// Mitsubishi GX Works2 project: PLC_Group24 (1)   PLC: FX3G

// global labels: Global1
VAR_GLOBAL
  X007_Stat_Work AT X007 : BOOL;  (* יום העבודה מתחיל בלחיצה על מתג X7 *)
  Y7_Day_Work AT Y007 : BOOL;  (* נורה Y7 תשאר דלוקה לאורך כל יום העבודה *)
  X5_Emergency_switch AT X005 : BOOL;  (* לחיצה על מתג חירום X5 *)
  input_Petel AT D1110 : REAL;  (* פטל(גרם),קלט כמות פתיחה{חומר גלם} *)
  linput_Lemon AT D1120 : REAL;  (* לימון(גרם), קלט כמות פתיחה{חומר גלם} *)
  input_Stabalized AT D1130 : REAL;  (* מייצבים(גרם), קלט כמות פתיחה{חומר גלם} *)
  input_Gummy_Bears AT D1140 : INT;  (* דובי גומי(יחידות), קלט כמות פתיחה{חומר גלם} *)
  X1_Stage1_start AT X001 : BOOL;  (* בלחיצה על המתג תתבצע דגימה של Analog Input1 ויבחר סוג הגומיגם. *)
END_VAR
VAR_GLOBAL CONSTANT
  Regular_Lower_limit : INT;  (* 0 ≤ input ≤ 5          נייצר גומיגם רגיל *)
  Regular_Upper_limit : INT := 5;  (* 0 ≤ input ≤ 5          נייצר גומיגם רגיל *)
  Treat_Lower_limit : INT := 6;  (* 6 ≤ input ≤ 10       נייצר גומיגם פינוק. *)
  Treat_Upper_limit : INT := 9;  (* 6 ≤ input ≤ 10       נייצר גומיגם פינוק. *)
  TABLE1_RegularPETAL_Lemon : REAL := 35;  (* טבלה 1 -        גלידה פטל רגיל -לימון   35 גרם *)
  TABLE1_RegularPETAL_Petel : REAL := 280;  (* טבלה 1 -          גלידה פטל רגיל -פטל 280 גרם *)
  TABLE1_RegularLemon_Petel : REAL;  (* טבלה 1 -        גלידה לימון רגיל -פטל     0 גרם *)
  TABLE1_RegularLemon_Lemon : REAL := 420;  (* טבלה 1 -     גלידה לימון רגיל -לימון 420 גרם *)
  TABLE1_RegularLemon_Stabalized : REAL := 70;  (* טבלה 1 - גלידה לימון רגיל -מייצבים   70 גרם *)
  TABLE1_TreatPETAL_Petel : REAL := 385;  (* טבלה 1 -          גלידה פטל פינוק -פטל 385 גרם *)
  TABLE1_TreatPETAL_Lemon : REAL := 105;  (* טבלה 1 -       גלידה פטל פינוק -לימון  105 גרם *)
  TABLE1_TreatPETAL_Stabalized : REAL := 70;  (* טבלה 1 -  גלידה פטל פינוק -מייצבים   70  גרם *)
  TABLE1_TreatLemon_Petel : REAL;  (* טבלה 1 -       גלידה לימון פינוק -פטל   0    גרם *)
  TABLE1_TreatLemon_Lemon : REAL := 560;  (* טבלה 1 -     גלידה לימון פינוק -לימון   560 גרם *)
  TABLE1_TreatLemon_Stabalized : REAL := 140;  (* טבלה 1 - גלידה לימון פינוק -מייצבים   140 גרם *)
END_VAR
VAR_GLOBAL
  amaount_Petel AT D1115 : REAL;  (* פטל(גרם),קלט כמות פתיחה{חומר גלם} *)
  amaount_Lemon AT D1125 : REAL;  (* לימון(גרם), קלט כמות פתיחה{חומר גלם} *)
  amaount_Stabalized AT D1135 : REAL;  (* מייצבים(גרם), קלט כמות פתיחה{חומר גלם} *)
  amaount_Gummy_Bears AT D1145 : INT;  (* דובי גומי(יחידות), קלט כמות פתיחה{חומר גלם} *)
  M110_Regular_Petel AT M110 : BOOL;  (* בוליאני,בדיקת כמות פטל לייצור גלידה  רגיל *)
  M230_Treat_Stabalized AT M230 : BOOL;  (* בוליאני,בדיקת כמות מייצבים לייצור גידה פינוק *)
  M220_Treat_Lemon AT M220 : BOOL;  (* בוליאני,בדיקת כמות לימון לייצור גלידה פינוק *)
  M210_Treat_Petel AT M210 : BOOL;  (* בוליאני,בדיקת כמות פטל לייצור גלידה פינוק *)
  M120_Regularl_Lemon AT M120 : BOOL;  (* בוליאני,בדיקת כמות לימון לייצור גלידה  רגיל *)
  M250_Treat_Can_produce AT M250 : BOOL;  (* בוליאני,האם יכול לייצור גלידה פינוק *)
END_VAR
VAR_GLOBAL CONSTANT
  TABLE1_RegularPETAL_Stabalized : REAL := 35;  (* טבלה 1 -   גלידה פטל רגיל -מייצבים   35 גרם *)
END_VAR
VAR_GLOBAL
  M140_Regularl_Gummy_Bears AT M140 : BOOL;  (* בוליאני,בדיקת כמות דובי גומי לייצור גלידה  רגיל *)
  M130_Regularl_Stabalized AT M130 : BOOL;  (* בוליאני,בדיקת כמות מיצבים לייצור גלידה  רגיל *)
  M240_Treat_Gummy_Bears AT M240 : BOOL;  (* בוליאני,בדיקת כמות דובי גומי לייצור גלידה פינוק *)
END_VAR
VAR_GLOBAL CONSTANT
  TABLE2_Regular_Gummy_Bears_gr : REAL := 28;  (* טבלה 2 -        גלידה פטל רגיל -דובי גומי   28 גרם *)
  TABLE2_Treat_Gummy_Bears_gr : REAL := 70;  (* טבלה 2 -      גלידה פטל פינוק -דובי גומי   70  גרם *)
END_VAR
VAR_GLOBAL
  M100_Regular AT M100 : BOOL;  (* בוליאני,לייצר גומיגם רגיל *)
  M101_Regular_Upper AT M101 : BOOL;  (* בוליאני,לייצר גומיגם רגיל-גבול עליון *)
  M102_Regular_Lower AT M102 : BOOL;  (* בוליאני,לייצר גומיגם רגיל-גבול תחתון *)
  M202_Treat_Lower AT M202 : BOOL;  (* בוליאני,לייצר גומיגם פינוק-גבול תחתון *)
  M200_Treat AT M200 : BOOL;  (* בוליאני,לייצר גומיגם פינוק *)
  M201_Treat_Upper AT M201 : BOOL;  (* בוליאני,לייצר גומיגם פינוק-גבול עליון *)
  M150_Regular_Can_produce AT M150 : BOOL;  (* בוליאני,האם יכול לייצור גלידה  רגיל *)
END_VAR
VAR_GLOBAL CONSTANT
  Analog_Input_divader : INT := 400;  (* Analog Input התאמת ערכי החיבור בחילוק ב400 *)
END_VAR
VAR_GLOBAL
  adj_analog_input_1 AT D1105 : INT;  (* דובי גומי(יחידות), קלט כמות פתיחה{חומר גלם} *)
  Y0_Ice_Cream_In_Process AT Y000 : BOOL;  (* הכנת הגלידה נמשכת 5 שניות במהלכן נורה Y0 דולקת. *)
  M_10_Not_Enough_Resources AT M10 : BOOL;  (* חסר חומר גלם - במידה ודולק יש לעצור מיידית את הייצור *)
  TS1_Coock_Ligth AT TS1 : BOOL;  (* בוליאני,האם יכול לייצור גלידה  רגיל *)
  TC1_stap1_cook_Ice_Cream AT TC1 : BOOL;  (* טיימר של 5 שניות,שלב 1 , של הכנת הגלידה *)
END_VAR
VAR_GLOBAL CONSTANT
  Time_cook_Ice_Cream : INT := 50;  (* 5 שניות של שלב ראשון של בישול הגלידה *)
END_VAR
VAR_GLOBAL
  Container_Ice_Cream_Petel AT D1150 : REAL;  (* מיכל ההכנה,גלידת פטל(גרם) כמויות, *)
  Container_Ice_Cream_Lemon AT D1160 : REAL;  (* מיכל ההכנה,גלידת לימון(גרם) כמויות *)
  Container_Cooling_Petel AT D1170 : REAL;  (* מיכל הקירור,גלידת פטל(גרם) כמויות *)
  Container_Cooling_Lemon AT D1180 : REAL;  (* מיכל הקירור,גלידת לימון(גרם) כמויות *)
  container_Mixing AT D1190 : REAL;  (* מיכל הערבוב של הגלידות ביחד עם גלידת הפט, גלידת הלימון, והגומיגם ביחד *)
END_VAR
VAR_GLOBAL CONSTANT
  Emptying_Container : REAL;  (* ריקון המיכל לאחר שהועבר למיכל אחר *)
END_VAR
VAR_GLOBAL
  X2_Stage2_start AT X002 : BOOL;  (* ע"י לחיצה על מתג X2 הגלידה תועבר ממכלי הכנת הטעמים למכלי הקירור (מכל נפרד עבור כל טעם) ותהליך הקירור מתחיל. *)
  Y2_step2_Cooling_In_Process AT Y002 : BOOL;  (* במהלך הקירור נורה 2Y דולקת. *)
  TS2_Cooling_Ligth AT TS2 : BOOL;  (* בוליאני,האם האם מקרר את הגלידה *)
  TC2_stap2_Cooling_Ice_Cream AT TC2 : BOOL;  (* משך קירור הגלידה הוא עד 8 שניות *)
END_VAR
VAR_GLOBAL CONSTANT
  Time_Cooling_Ice_Cream : INT := 80;  (* משך קירור הגלידה הוא עד 8 שניות *)
END_VAR
VAR_GLOBAL
  X3_High_temp_switch AT X003 : BOOL;  (* או עד שחיישן הטמפרטורה X3 מצביע על טמפרטורה של 10 מעלות ומטה. *)
  Y5_step3_Mixing_In_Progress AT Y005 : BOOL;  (* משך הערבוב תלוי בסוג הגומיגם, ניתן לראות טבלה 3. בזמן הערבוב נורות Y5 ו-Y6 מהבהבות לסירוגין *)
  Y6_step3_Mixing_In_Progress AT Y006 : BOOL;  (* משך הערבוב תלוי בסוג הגומיגם, ניתן לראות טבלה 3. בזמן הערבוב נורות Y5 ו-Y6 מהבהבות לסירוגין *)
  M56_Flashing_Intermittently_Y5_6 AT M56 : BOOL;  (* בוליאני של הבהוב הורות Y5 ו- Y6 *)
  Step3_Mixing_Time AT D1300 : INT;  (* מקבל בהתאם את הערך הרצוי מטבלה 3 - בהתאם לסוג הגומיגם שייצרנו *)
  TS4_Flashing_Ligth1 AT TS4 : BOOL;  (* בוליאני,האם האם מערבב - 2 *)
  TC4_stap3_Mixing1 AT TC4 : BOOL;  (* משך קירור הגלידה הוא ערבוב תלוי בסוג הגומיגם לפי טבלה 3 *)
  TS5_Flashing_Ligth2 AT TS5 : BOOL;  (* בוליאני,האם האם מערבב - 2 *)
  TC5_stap3_Mixing2 AT TC5 : BOOL;  (* משך קירור הגלידה הוא ערבוב תלוי בסוג הגומיגם לפי טבלה 3 *)
END_VAR
VAR_GLOBAL CONSTANT
  TABLE2_Regular_Gummy_Bears_unit : INT := 28;  (* טבלה 2 -        גלידה פטל רגיל -דובי גומי   28 גרם *)
  TABLE2_Treat_Gummy_Bears_unit : INT := 70;  (* טבלה 2 -      גלידה פטל פינוק -דובי גומי   70  גרם *)
  TABLE3_Treat_Mixing_time : INT := 50;  (* טבלה 3- משך זמן הערבוב (5 שניות) כתלות בסוג הגומיגם (פינוק) *)
  TABLE3_Regular_Mixing_time : INT := 30;  (* טבלה 3- משך זמן הערבוב (3 שניות) כתלות בסוג הגומיגם (רגיל) *)
END_VAR
VAR_GLOBAL
  M300_Stage3_Sart AT M300 : BOOL;  (* התחל שלב 3 , סיום שלב 2 *)
  X4_Stage4_start AT X004 : BOOL;  (* שלב 4 	תהליך זה יתחיל ע"י הרמת מתג X4. *)
  X0_One_Cone_package AT X000 : BOOL;  (* עבור אריזת גביע גומיגם בודד יש להרים את מתג X0. *)
  Y4_step4_Pakage_7Cone_in_process AT Y004 : BOOL;  (* •	בסיום אריזת הגביע הראשון במארז, יש להדליק את נורה Y4, ובסיום אריזת המארז נורה Y4 תיכבה. *)
END_VAR
VAR_GLOBAL CONSTANT
  Step3_flashing_switch : INT := 1;  (* מקבל בהתאם את הערך הרצוי מטבלה 3 - בהתאם לסוג הגומיגם שייצרנו *)
END_VAR
VAR_GLOBAL
  TS3_Micing_time AT TS3 : BOOL;  (* בוליאני,האם האם מערבב - 2 *)
  TC3_stap3_Mixing AT TC3 : BOOL;  (* משך קירור הגלידה הוא ערבוב תלוי בסוג הגומיגם לפי טבלה 3 *)
END_VAR
VAR_GLOBAL CONSTANT
  Step4_count_7cones : INT := 7;  (* ספירה של 7 גביעים באריזת הגומיגם *)
  Step4_count_First_cones : INT := 1;  (* ספירה של ביע הראשון שנכנס לאירזה *)
END_VAR
VAR_GLOBAL
  CC1_count_First_Cones AT CC1 : BOOL;  (* ספירה של 1 גביעי גלידה *)
  CC0_count_7Cones AT CC0 : BOOL;  (* ספירה של 7 גביעי גלידה *)
  CS1_count_first_cone AT CS1 : BOOL;  (* ספירה של 1 גביעי גלידה *)
  CS0_count_7_cone AT CS0 : BOOL;  (* ספירה של 7 גביעי גלידה *)
END_VAR
VAR_GLOBAL CONSTANT
  Add_one_pack : INT := 1;  (* הוספת אריזה אחת לכמות באחסון *)
  Tourn_false : BOOL;  (* הפיכת המשתנים ל-FFALSE *)
  table2_Regular_1cone_Total_grams : REAL := 124;  (* כמות הגרם הנדרשת ליחידת גומיגם רגיל אחד (124גרם) *)
  table2_Treat_1cone_Total_grams : REAL := 190;  (* כמות הגרם הנדרשת ליחידת גומיגם רגיל אחד (190גרם) *)
  New_day_Storage_is_empty : INT;  (* יום חדש, "כל המשתנים יתאפסו וניתן יהיה להתחיל יום עבודה מחדש בלחיצה נוספת על מתג X7. " *)
END_VAR
VAR_GLOBAL
  Analog_Input_1 AT D8280 : INT;  (* Analog Input 1 – D8280 --> סוג הגומיגם יבחר כתלות בערך *)
  AnalogOutput AT D8282 : INT;  (* Analog Output – D8282 --> מספר מארזי הגומיגם שיוצרו במהלך היום ביחידות עשרוניות *)
  Total_Packs AT D1100 : INT;
END_VAR
VAR_GLOBAL CONSTANT
  adj_amaunt_Packs_To_AnalogOutpot : INT := 40;  (* הערך המותאם ליציאה האנלוגית(בהכפלה ב40) *)
END_VAR
VAR_GLOBAL
  M_20_Not_Enough_Resources AT M20 : BOOL;  (* חסר חומר גלם - שלב 4 , במידה ודולק יש לעצור מיידית את הייצור *)
END_VAR

// task Task_01 (event TRUE, interval 0, priority 31): POU_01

PROGRAM POU_01
(* structured ladder/FBD written out as ST: instructions are called as NAME(EN, inputs, outputs); _pN, _eN, _tN stand for wires *)
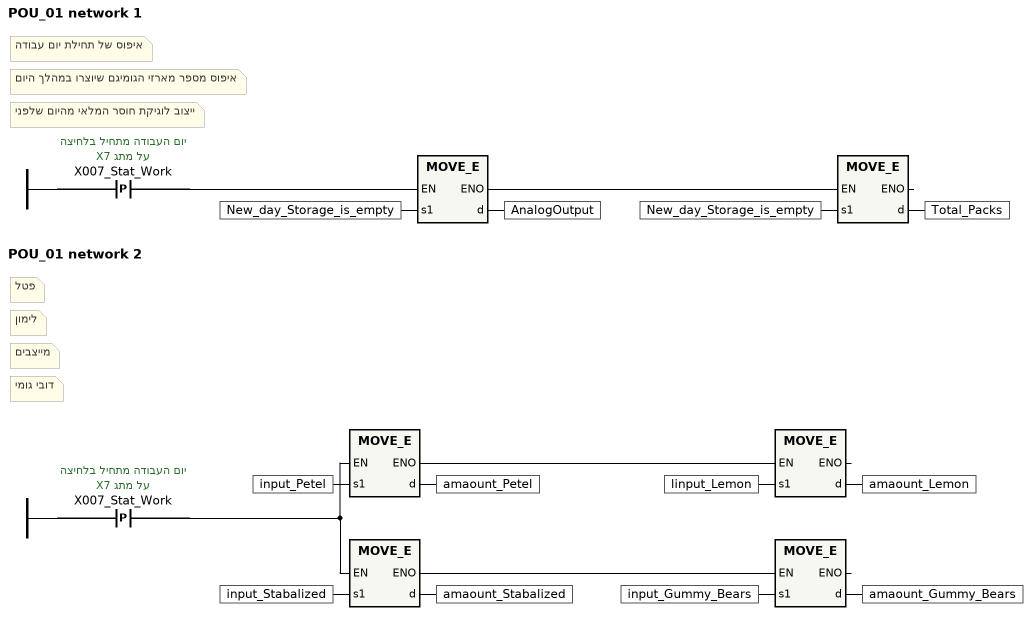
(* network 1 איפוס תחילת יום *)
(* איפוס של תחילת יום עבודה *)
(* איפוס מספר מארזי הגומיגם שיוצרו במהלך היום *)
(* ייצוב לוגיקת חוסר המלאי מהיום שלפני *)
_e1 := MOVE_E(LDP(TRUE, X007_Stat_Work), New_day_Storage_is_empty, AnalogOutput);
MOVE_E(_e1, New_day_Storage_is_empty, Total_Packs);
(* network 2 הזנת מלאי לערכים *)
(* פטל *)
(* לימון *)
(* מייצבים *)
(* דובי גומי *)
_p1 := LDP(TRUE, X007_Stat_Work);
_e2 := MOVE_E(_p1, input_Petel, amaount_Petel);
MOVE_E(_e2, linput_Lemon, amaount_Lemon);
_e3 := MOVE_E(_p1, input_Stabalized, amaount_Stabalized);
MOVE_E(_e3, input_Gummy_Bears, amaount_Gummy_Bears);
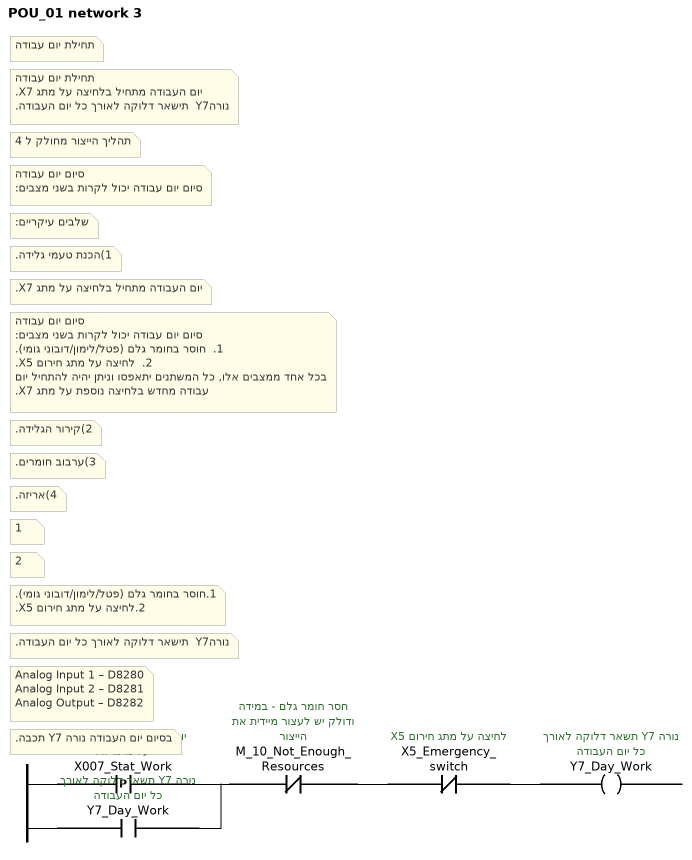
(* network 3 תחילת/סיום יום עבודה *)
(* תחילת יום עבודה *)
(* תחילת יום עבודה / יום העבודה מתחיל בלחיצה על מתג X7.   / נורהY7  תישאר דלוקה לאורך כל יום העבודה. *)
(* תהליך הייצור מחולק ל 4 *)
(* סיום יום עבודה / סיום יום עבודה יכול לקרות בשני מצבים: *)
(* שלבים עיקריים: *)
(* 1)הכנת טעמי גלידה. *)
(* יום העבודה מתחיל בלחיצה על מתג X7. *)
(* סיום יום עבודה / סיום יום עבודה יכול לקרות בשני מצבים: / 1.	חוסר בחומר גלם (פטל/לימון/דובוני גומי). / 2.	לחיצה על מתג חירום X5.  / בכל אחד ממצבים אלו, כל המשתנים יתאפסו וניתן יהיה להתחיל יום עבודה מחדש בלחיצה נוספת על מתג X7. *)
(* 2)קירור הגלידה. *)
(* 3)ערבוב חומרים. *)
(* 4)אריזה. *)
(* 1 *)
(* 2 *)
(* 1.חוסר בחומר גלם (פטל/לימון/דובוני גומי). / 2.לחיצה על מתג חירום X5. *)
(* נורהY7  תישאר דלוקה לאורך כל יום העבודה. *)
(* Analog Input 1 – D8280 / Analog Input 2 – D8281 / Analog Output – D8282 *)
(* בסיום יום העבודה נורה Y7 תכבה. *)
Y7_Day_Work := ((LDP(TRUE, X007_Stat_Work) OR Y7_Day_Work) AND NOT M_10_Not_Enough_Resources) AND NOT X5_Emergency_switch;
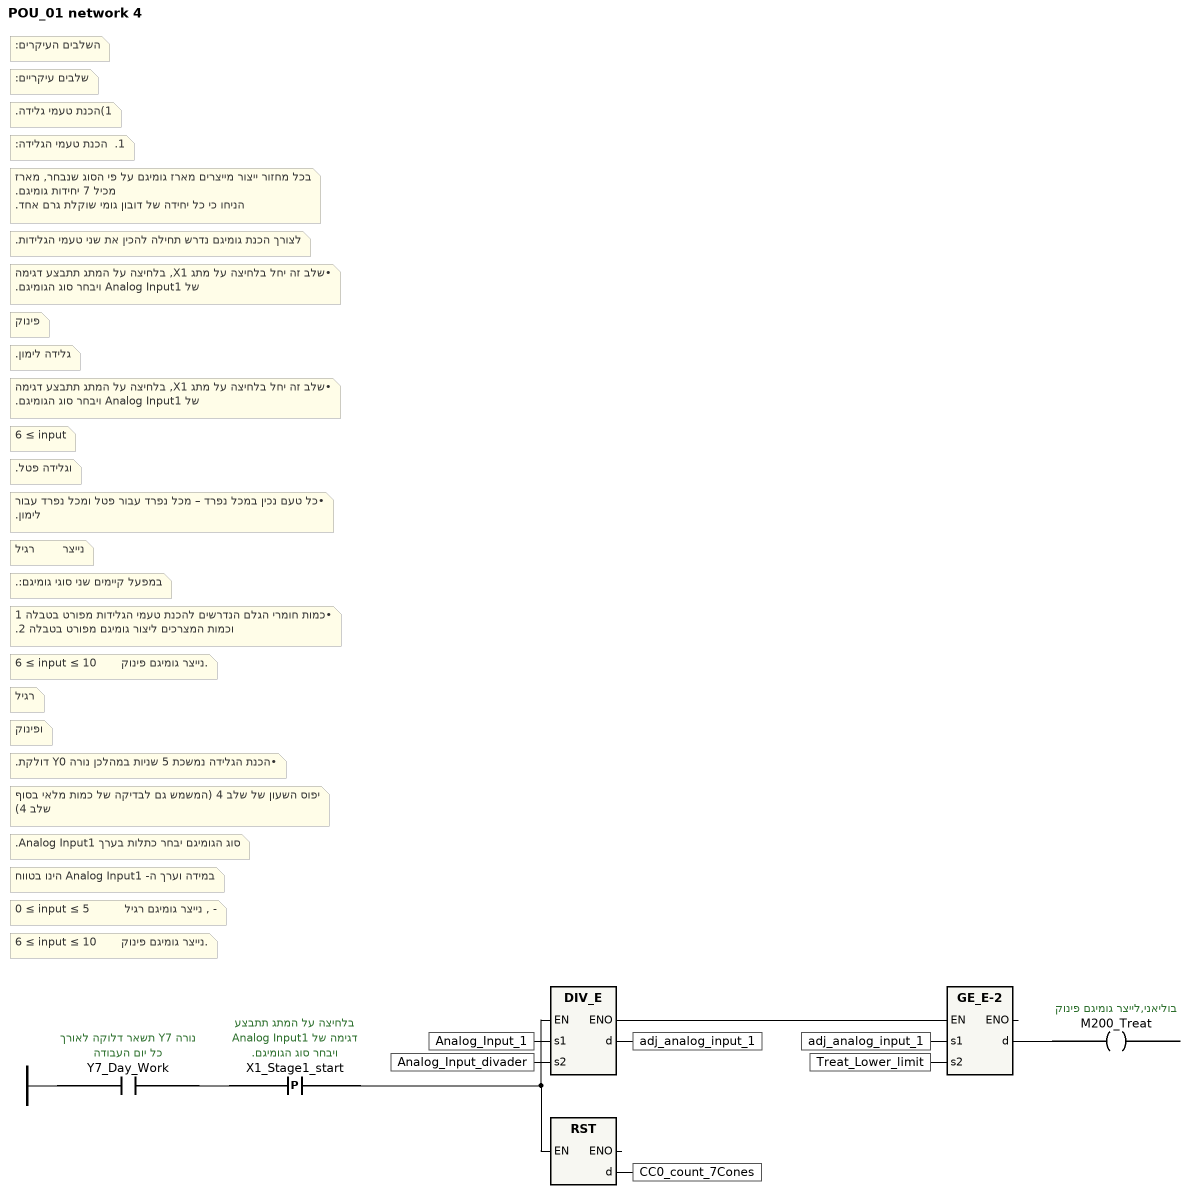
(* network 4 תחילה ובחירת סוג *)
(* השלבים העיקרים: *)
(* שלבים עיקריים: *)
(* 1)הכנת טעמי גלידה. *)
(* 1.	הכנת טעמי הגלידה: *)
(* בכל מחזור ייצור מייצרים מארז גומיגם על פי הסוג שנבחר, מארז מכיל 7 יחידות גומיגם.  / הניחו כי כל יחידה של דובון גומי שוקלת גרם אחד. *)
(* לצורך הכנת גומיגם נדרש תחילה להכין את שני טעמי הגלידות. *)
(* •שלב זה יחל בלחיצה על מתג X1, בלחיצה על המתג תתבצע דגימה של Analog Input1 ויבחר סוג הגומיגם. *)
(* פינוק *)
(* גלידה לימון. *)
(* •שלב זה יחל בלחיצה על מתג X1, בלחיצה על המתג תתבצע דגימה של Analog Input1 ויבחר סוג הגומיגם. *)
(* 6 ≤ input *)
(* וגלידה פטל. *)
(* •כל טעם נכין במכל נפרד – מכל נפרד עבור פטל ומכל נפרד עבור לימון. *)
(* נייצר        רגיל *)
(* במפעל קיימים שני סוגי גומיגם:. *)
(* •כמות חומרי הגלם הנדרשים להכנת טעמי הגלידות מפורט בטבלה 1 וכמות המצרכים ליצור גומיגם מפורט בטבלה 2. *)
(* 6 ≤ input ≤ 10       נייצר גומיגם פינוק. *)
(* רגיל *)
(* ופינוק *)
(* •הכנת הגלידה נמשכת 5 שניות במהלכן נורה Y0 דולקת. *)
(* יפוס השעון של שלב 4 (המשמש גם לבדיקה של כמות מלאי בסוף שלב 4) *)
(* סוג הגומיגם יבחר כתלות בערך Analog Input1. *)
(* במידה וערך ה- Analog Input1 הינו בטווח *)
(* 0 ≤ input ≤ 5          נייצר גומיגם רגיל , - *)
(* 6 ≤ input ≤ 10       נייצר גומיגם פינוק. *)
_p1 := Y7_Day_Work AND LDP(TRUE, X1_Stage1_start);
_e2 := DIV_E(_p1, Analog_Input_1, Analog_Input_divader, adj_analog_input_1);
GE_E(_e2, adj_analog_input_1, Treat_Lower_limit, _t3);
M200_Treat := _t3;
RST(_p1, CC0_count_7Cones);
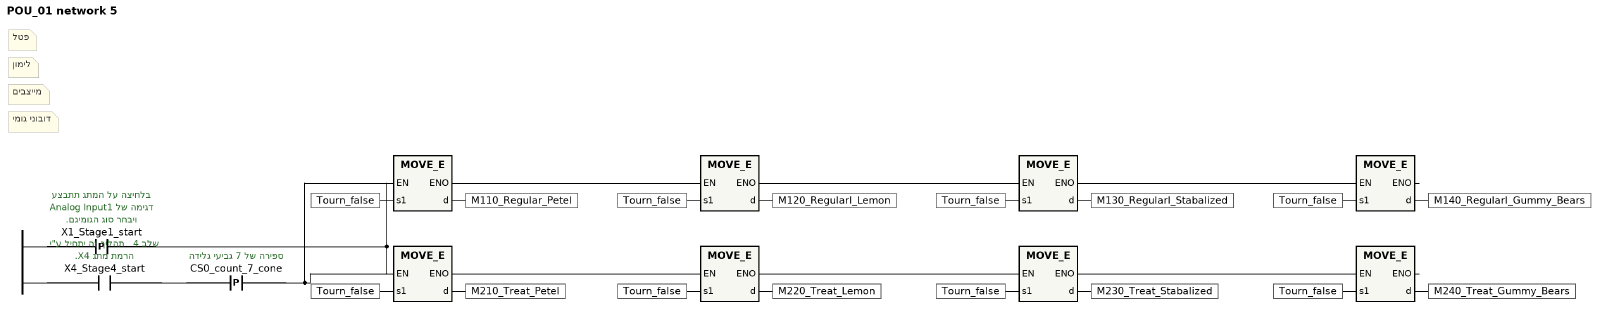
(* network 5 *)
(* פטל *)
(* לימון *)
(* מייצבים *)
(* דובוני גומי *)
_p1 := LDP(TRUE, X1_Stage1_start) OR (X4_Stage4_start AND LDP(TRUE, CS0_count_7_cone));
_e2 := MOVE_E(_p1, Tourn_false, M110_Regular_Petel);
_e3 := MOVE_E(_e2, Tourn_false, M120_Regularl_Lemon);
_e4 := MOVE_E(_e3, Tourn_false, M130_Regularl_Stabalized);
MOVE_E(_e4, Tourn_false, M140_Regularl_Gummy_Bears);
_e5 := MOVE_E(_p1, Tourn_false, M210_Treat_Petel);
_e6 := MOVE_E(_e5, Tourn_false, M220_Treat_Lemon);
_e7 := MOVE_E(_e6, Tourn_false, M230_Treat_Stabalized);
MOVE_E(_e7, Tourn_false, M240_Treat_Gummy_Bears);
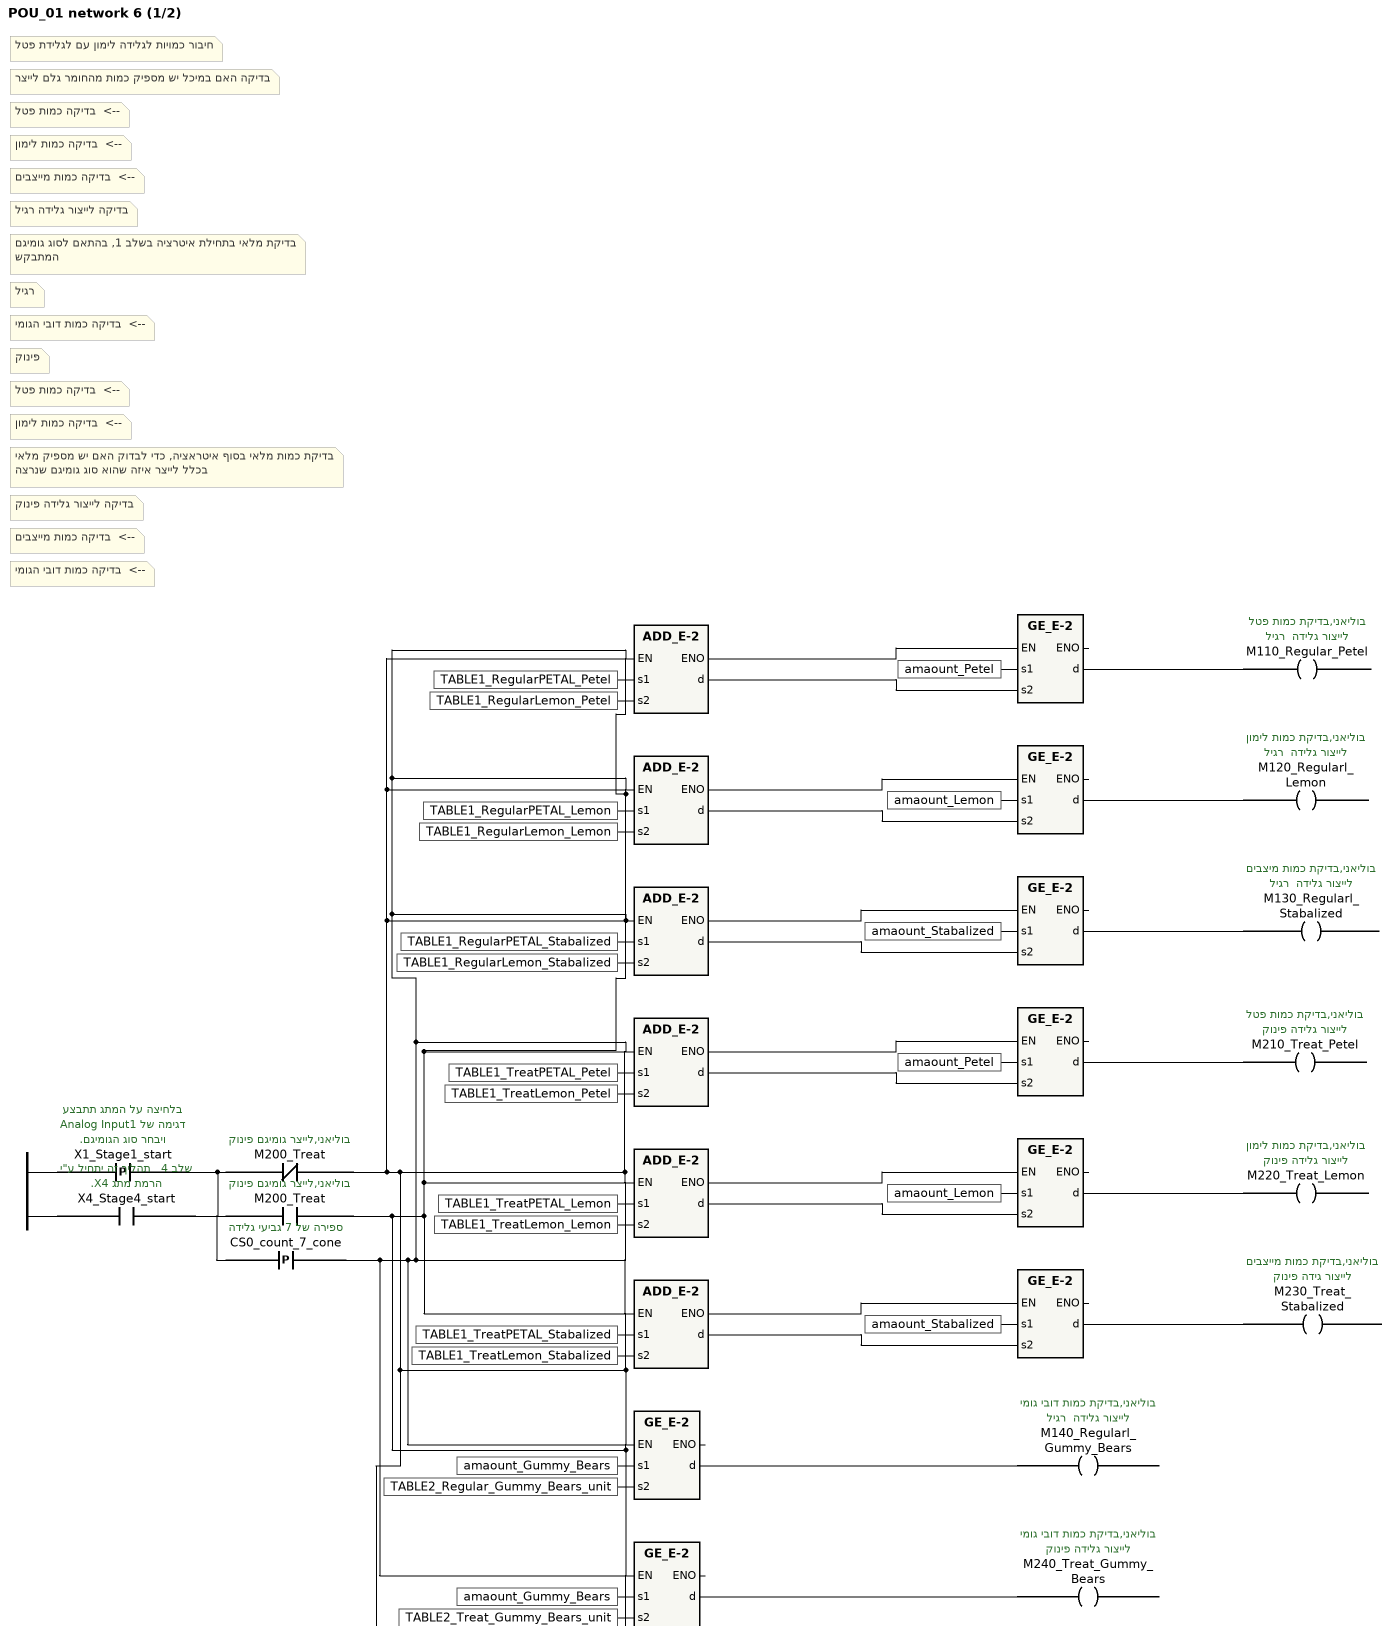
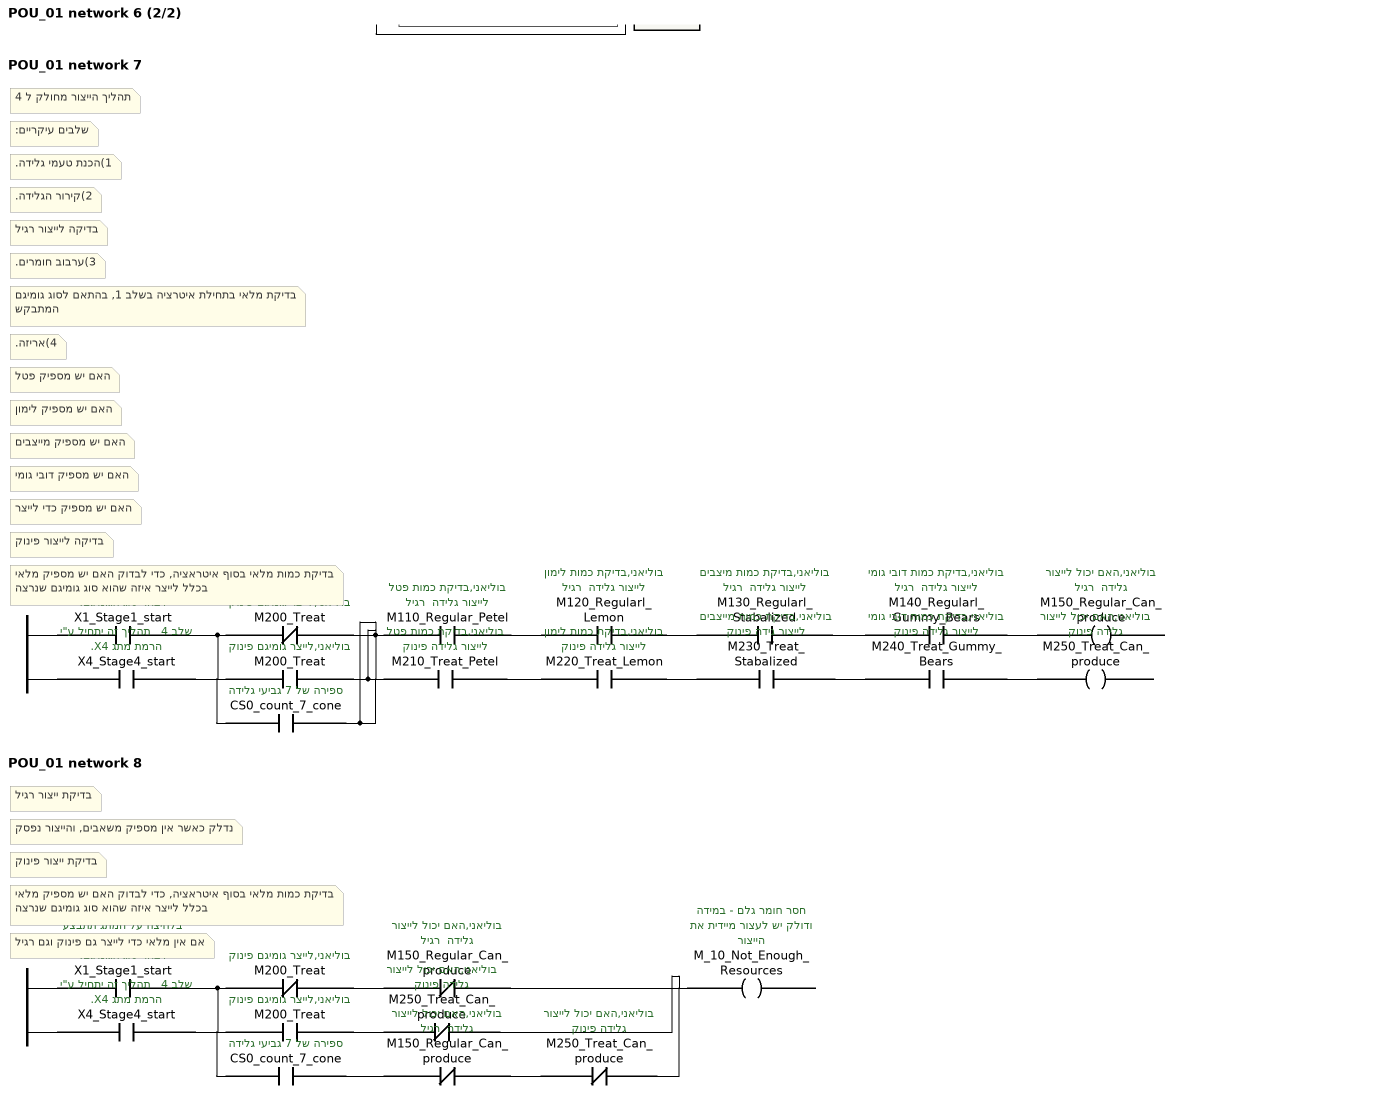
(* network 6 *)
(* חיבור כמויות לגלידה לימון עם לגלידת פטל *)
(* בדיקה האם במיכל יש מספיק כמות מהחומר גלם לייצר *)
(* -->  בדיקה כמות פטל *)
(* -->  בדיקה כמות לימון *)
(* -->  בדיקה כמות מייצבים *)
(* בדיקה לייצור גלידה רגיל *)
(* בדיקת מלאי בתחילת איטרציה בשלב 1, בהתאם לסוג גומיגם המתבקש *)
(* רגיל *)
(* -->  בדיקה כמות דובי הגומי *)
(* פינוק *)
(* -->  בדיקה כמות פטל *)
(* -->  בדיקה כמות לימון *)
(* בדיקת כמות מלאי בסוף איטראציה, כדי לבדוק האם יש מספיק מלאי בכלל לייצר איזה שהוא סוג גומיגם שנרצה *)
(* בדיקה לייצור גלידה פינוק *)
(* -->  בדיקה כמות מייצבים *)
(* -->  בדיקה כמות דובי הגומי *)
_p1 := LDP(TRUE, X1_Stage1_start);
_p2 := (_p1 AND NOT M200_Treat) OR (_p1 AND M200_Treat) OR (X4_Stage4_start AND LDP(TRUE, CS0_count_7_cone));
_e4 := ADD_E(_p2, TABLE1_RegularPETAL_Petel, TABLE1_RegularLemon_Petel, _t3);
GE_E(_e4, amaount_Petel, _t3, _t5);
M110_Regular_Petel := _t5;
_e7 := ADD_E(_p2, TABLE1_RegularPETAL_Lemon, TABLE1_RegularLemon_Lemon, _t6);
GE_E(_e7, amaount_Lemon, _t6, _t8);
M120_Regularl_Lemon := _t8;
_e10 := ADD_E(_p2, TABLE1_RegularPETAL_Stabalized, TABLE1_RegularLemon_Stabalized, _t9);
GE_E(_e10, amaount_Stabalized, _t9, _t11);
M130_Regularl_Stabalized := _t11;
GE_E(_p2, amaount_Gummy_Bears, TABLE2_Regular_Gummy_Bears_unit, _t12);
M140_Regularl_Gummy_Bears := _t12;
_e14 := ADD_E(_p2, TABLE1_TreatPETAL_Petel, TABLE1_TreatLemon_Petel, _t13);
GE_E(_e14, amaount_Petel, _t13, _t15);
M210_Treat_Petel := _t15;
_e17 := ADD_E(_p2, TABLE1_TreatPETAL_Lemon, TABLE1_TreatLemon_Lemon, _t16);
GE_E(_e17, amaount_Lemon, _t16, _t18);
M220_Treat_Lemon := _t18;
_e20 := ADD_E(_p2, TABLE1_TreatPETAL_Stabalized, TABLE1_TreatLemon_Stabalized, _t19);
GE_E(_e20, amaount_Stabalized, _t19, _t21);
M230_Treat_Stabalized := _t21;
GE_E(_p2, amaount_Gummy_Bears, TABLE2_Treat_Gummy_Bears_unit, _t22);
M240_Treat_Gummy_Bears := _t22;
(* network 7 *)
(* תהליך הייצור מחולק ל 4 *)
(* שלבים עיקריים: *)
(* 1)הכנת טעמי גלידה. *)
(* 2)קירור הגלידה. *)
(* בדיקה לייצור רגיל *)
(* 3)ערבוב חומרים. *)
(* בדיקת מלאי בתחילת איטרציה בשלב 1, בהתאם לסוג גומיגם המתבקש *)
(* 4)אריזה. *)
(* האם יש מספיק פטל *)
(* האם יש מספיק לימון *)
(* האם יש מספיק מייצבים *)
(* האם יש מספיק דובי גומי *)
(* האם יש מספיק כדי לייצר *)
(* בדיקה לייצור פינוק *)
(* בדיקת כמות מלאי בסוף איטראציה, כדי לבדוק האם יש מספיק מלאי בכלל לייצר איזה שהוא סוג גומיגם שנרצה *)
_p1 := (X1_Stage1_start AND NOT M200_Treat) OR (X1_Stage1_start AND M200_Treat) OR (X4_Stage4_start AND CS0_count_7_cone);
M150_Regular_Can_produce := _p1 AND M110_Regular_Petel AND M120_Regularl_Lemon AND M130_Regularl_Stabalized AND M140_Regularl_Gummy_Bears;
M250_Treat_Can_produce := _p1 AND M210_Treat_Petel AND M220_Treat_Lemon AND M230_Treat_Stabalized AND M240_Treat_Gummy_Bears;
(* network 8 *)
(* בדיקת ייצור רגיל *)
(* נדלק כאשר אין מספיק משאבים, והייצור נפסק *)
(* בדיקת ייצור פינוק *)
(* בדיקת כמות מלאי בסוף איטראציה, כדי לבדוק האם יש מספיק מלאי בכלל לייצר איזה שהוא סוג גומיגם שנרצה *)
(* אם אין מלאי כדי לייצר גם פינוק וגם רגיל *)
M_10_Not_Enough_Resources := (X1_Stage1_start AND NOT M200_Treat AND NOT M150_Regular_Can_produce) OR (X1_Stage1_start AND M200_Treat AND NOT M250_Treat_Can_produce) OR (X4_Stage4_start AND CS0_count_7_cone AND NOT M150_Regular_Can_produce AND NOT M250_Treat_Can_produce);
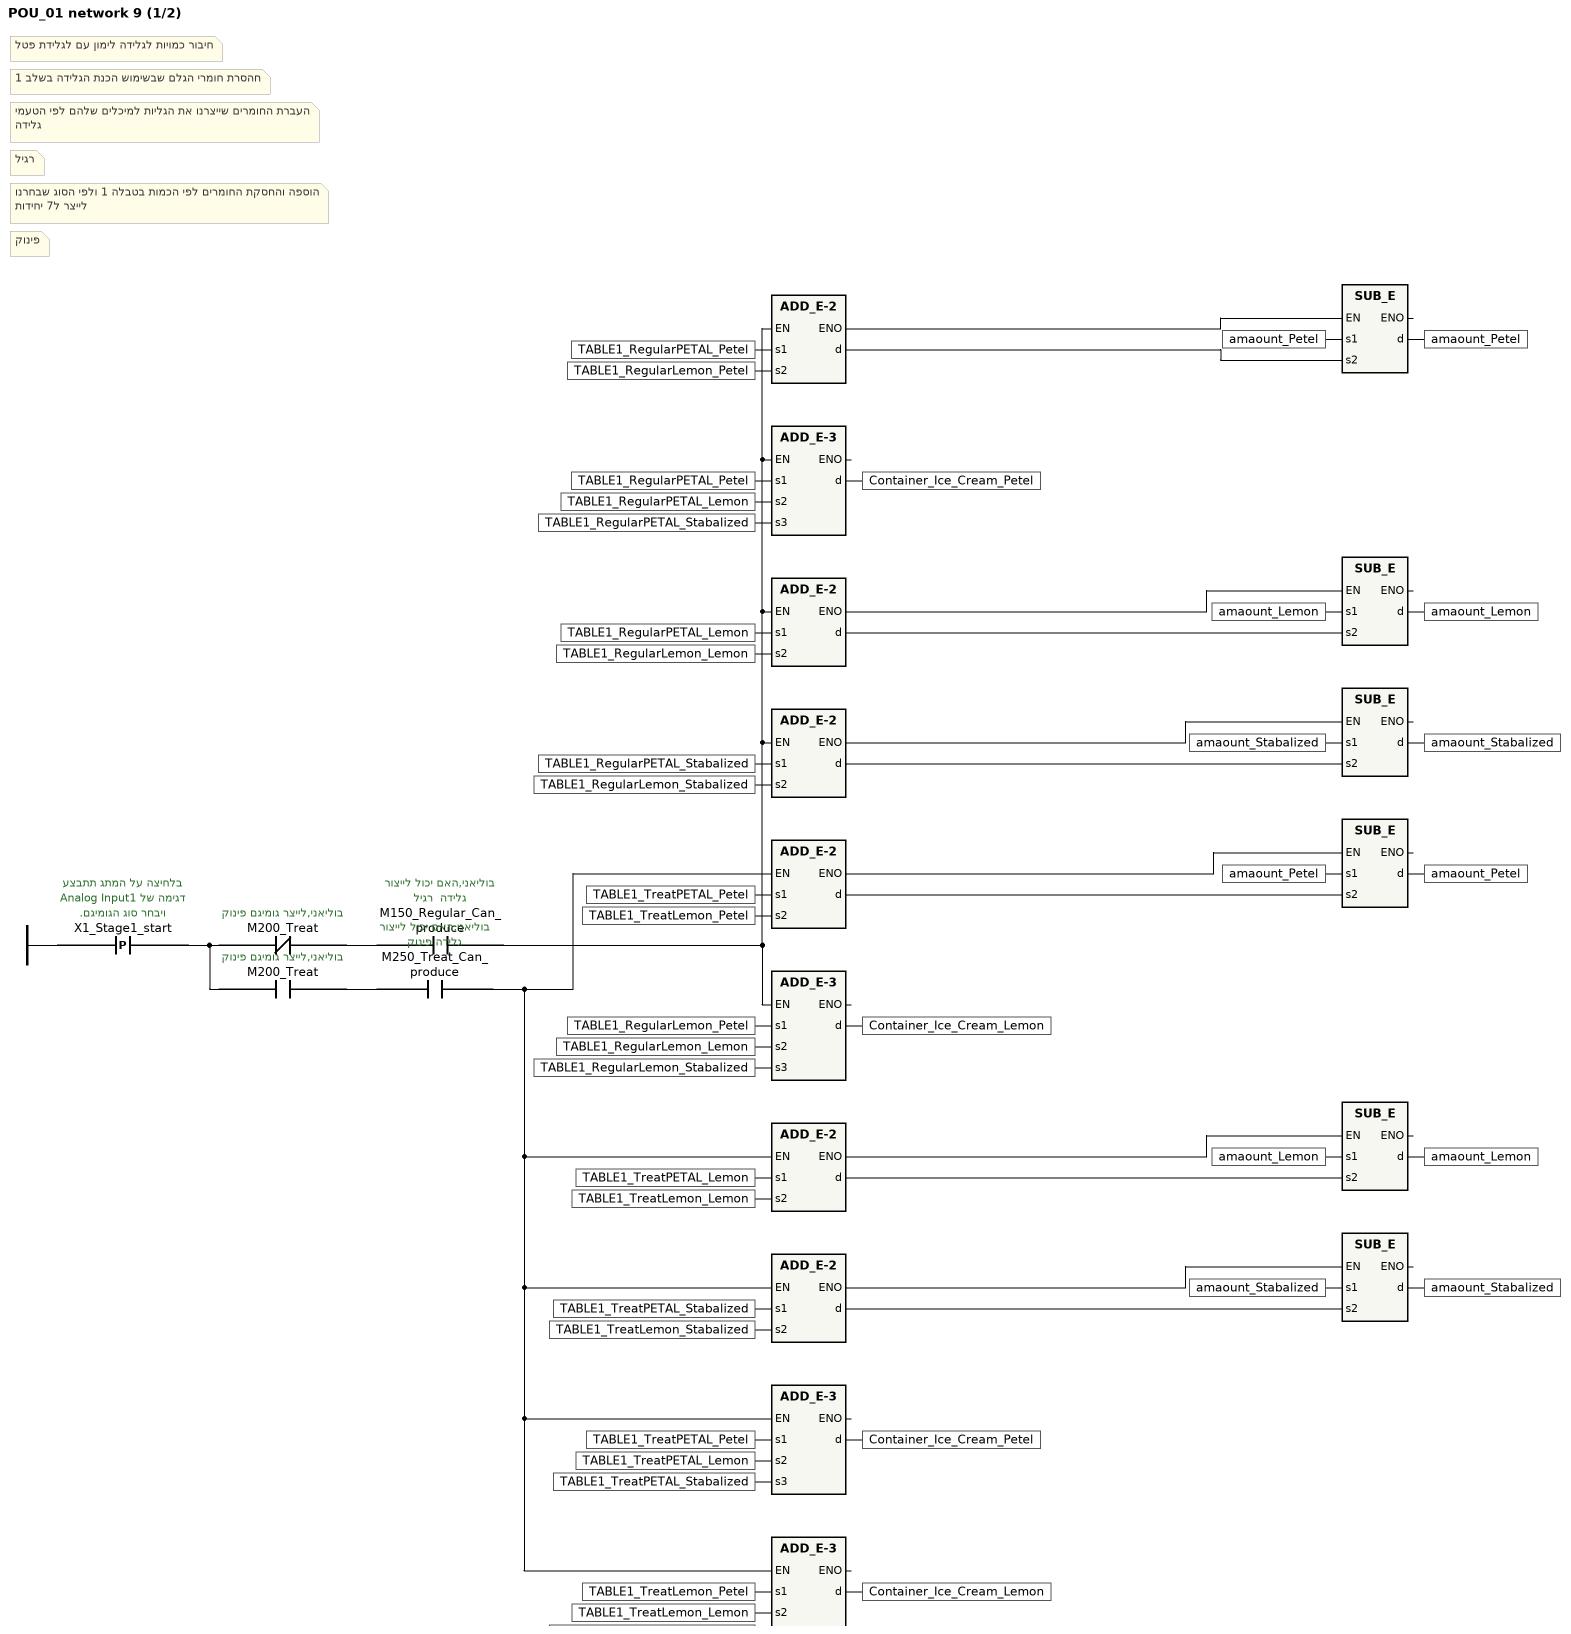
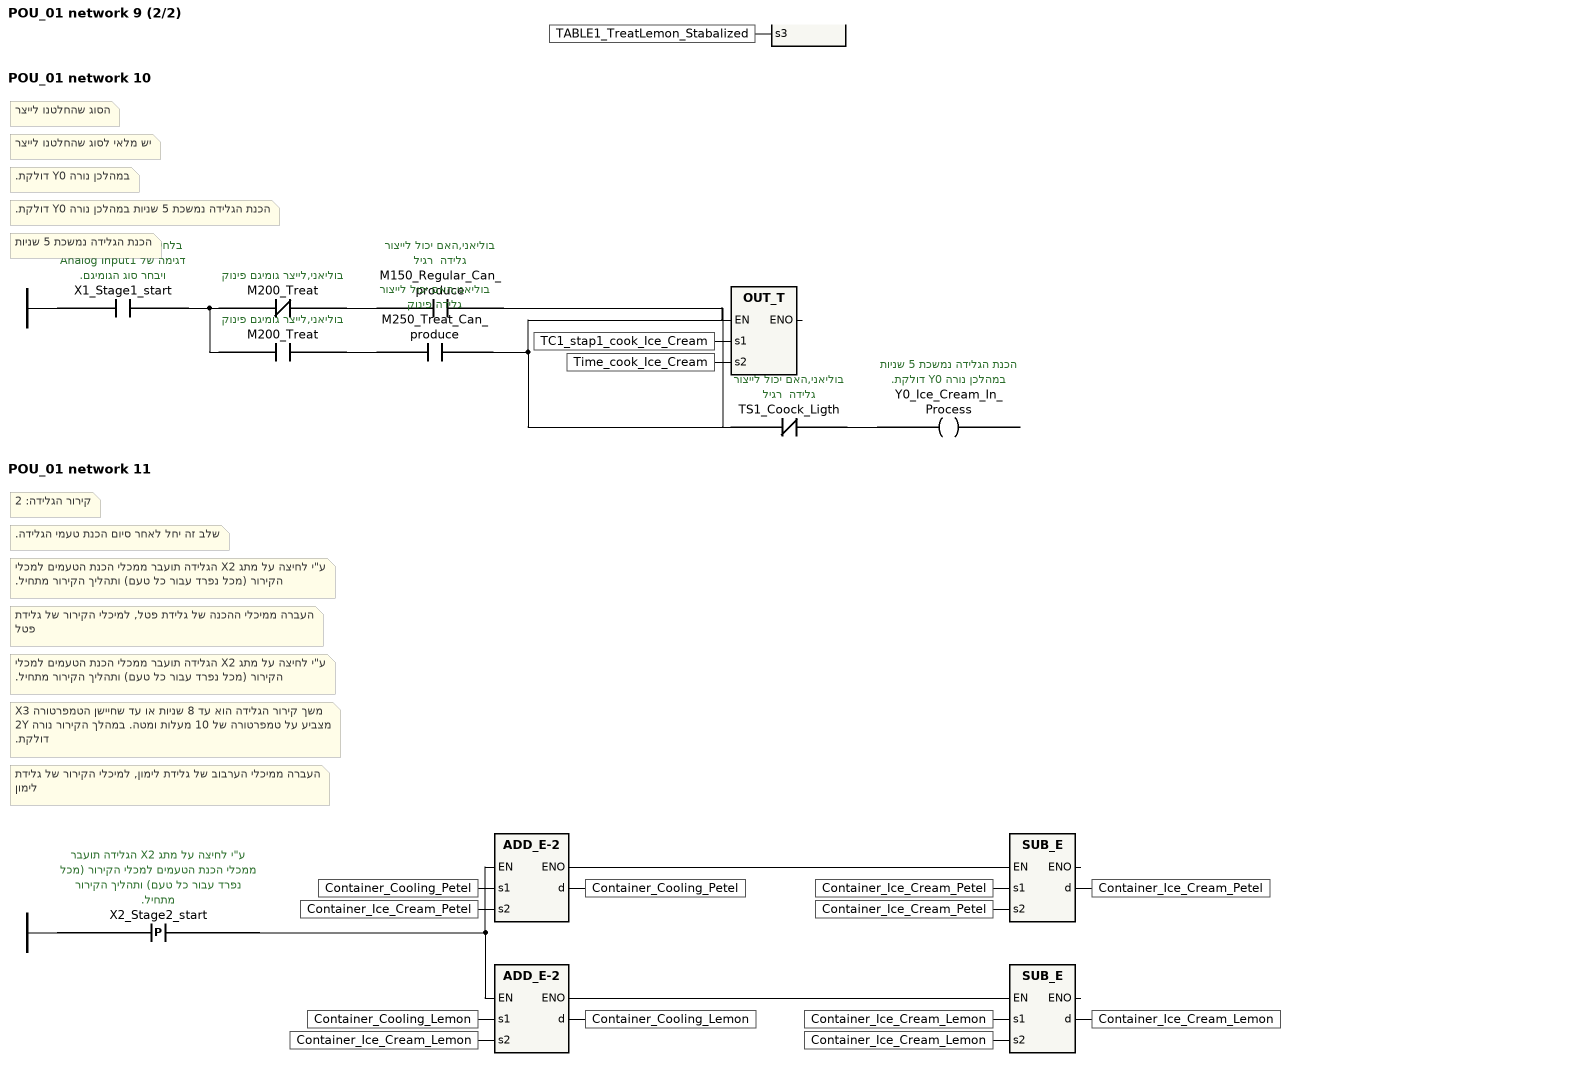
(* network 9 *)
(* חיבור כמויות לגלידה לימון עם לגלידת פטל *)
(* חהסרת חומרי הגלם שבשימוש הכנת הגלידה בשלב 1 *)
(* העברת החומרים שייצרנו את הגליות למיכלים שלהם לפי הטעמי גלידה *)
(* רגיל *)
(* הוספה והחסקת החומרים לפי הכמות בטבלה 1 ולפי הסוג שבחרנו לייצר ל7 יחידות *)
(* פינוק *)
_p1 := LDP(TRUE, X1_Stage1_start);
_p2 := _p1 AND NOT M200_Treat AND M150_Regular_Can_produce;
_e4 := ADD_E(_p2, TABLE1_RegularPETAL_Petel, TABLE1_RegularLemon_Petel, _t3);
SUB_E(_e4, amaount_Petel, _t3, amaount_Petel);
ADD_E(_p2, TABLE1_RegularPETAL_Petel, TABLE1_RegularPETAL_Lemon, TABLE1_RegularPETAL_Stabalized, Container_Ice_Cream_Petel);
_e6 := ADD_E(_p2, TABLE1_RegularPETAL_Lemon, TABLE1_RegularLemon_Lemon, _t5);
SUB_E(_e6, amaount_Lemon, _t5, amaount_Lemon);
ADD_E(_p2, TABLE1_RegularLemon_Petel, TABLE1_RegularLemon_Lemon, TABLE1_RegularLemon_Stabalized, Container_Ice_Cream_Lemon);
_e8 := ADD_E(_p2, TABLE1_RegularPETAL_Stabalized, TABLE1_RegularLemon_Stabalized, _t7);
SUB_E(_e8, amaount_Stabalized, _t7, amaount_Stabalized);
_p9 := _p1 AND M200_Treat AND M250_Treat_Can_produce;
_e11 := ADD_E(_p9, TABLE1_TreatPETAL_Petel, TABLE1_TreatLemon_Petel, _t10);
SUB_E(_e11, amaount_Petel, _t10, amaount_Petel);
ADD_E(_p9, TABLE1_TreatPETAL_Petel, TABLE1_TreatPETAL_Lemon, TABLE1_TreatPETAL_Stabalized, Container_Ice_Cream_Petel);
_e13 := ADD_E(_p9, TABLE1_TreatPETAL_Lemon, TABLE1_TreatLemon_Lemon, _t12);
SUB_E(_e13, amaount_Lemon, _t12, amaount_Lemon);
ADD_E(_p9, TABLE1_TreatLemon_Petel, TABLE1_TreatLemon_Lemon, TABLE1_TreatLemon_Stabalized, Container_Ice_Cream_Lemon);
_e15 := ADD_E(_p9, TABLE1_TreatPETAL_Stabalized, TABLE1_TreatLemon_Stabalized, _t14);
SUB_E(_e15, amaount_Stabalized, _t14, amaount_Stabalized);
(* network 10 *)
(* הסוג שהחלטנו לייצר *)
(* יש מלאי לסוג שהחלטנו לייצר *)
(* במהלכן נורה Y0 דולקת. *)
(* הכנת הגלידה נמשכת 5 שניות במהלכן נורה Y0 דולקת. *)
(* הכנת הגלידה נמשכת 5 שניות *)
_p1 := (X1_Stage1_start AND NOT M200_Treat AND M150_Regular_Can_produce) OR (X1_Stage1_start AND M200_Treat AND M250_Treat_Can_produce);
Y0_Ice_Cream_In_Process := _p1 AND NOT TS1_Coock_Ligth;
OUT_T(_p1, TC1_stap1_cook_Ice_Cream, Time_cook_Ice_Cream);
(* network 11 שלב 2 *)
(* קירור הגלידה: 2 *)
(* שלב זה יחל לאחר סיום הכנת טעמי הגלידה. *)
(* ע"י לחיצה על מתג X2 הגלידה תועבר ממכלי הכנת הטעמים למכלי הקירור (מכל נפרד עבור כל טעם) ותהליך הקירור מתחיל. *)
(* העברה ממיכלי ההכנה של גלידת פטל, למיכלי הקירור של גלידת פטל *)
(* ע"י לחיצה על מתג X2 הגלידה תועבר ממכלי הכנת הטעמים למכלי הקירור (מכל נפרד עבור כל טעם) ותהליך הקירור מתחיל. *)
(* משך קירור הגלידה הוא עד 8 שניות או עד שחיישן הטמפרטורה X3 מצביע על טמפרטורה של 10 מעלות ומטה. במהלך הקירור נורה 2Y דולקת. *)
(* העברה ממיכלי הערבוב של גלידת לימון, למיכלי הקירור של גלידת לימון *)
_p1 := LDP(TRUE, X2_Stage2_start);
_e2 := ADD_E(_p1, Container_Cooling_Petel, Container_Ice_Cream_Petel, Container_Cooling_Petel);
SUB_E(_e2, Container_Ice_Cream_Petel, Container_Ice_Cream_Petel, Container_Ice_Cream_Petel);
_e3 := ADD_E(_p1, Container_Cooling_Lemon, Container_Ice_Cream_Lemon, Container_Cooling_Lemon);
SUB_E(_e3, Container_Ice_Cream_Lemon, Container_Ice_Cream_Lemon, Container_Ice_Cream_Lemon);
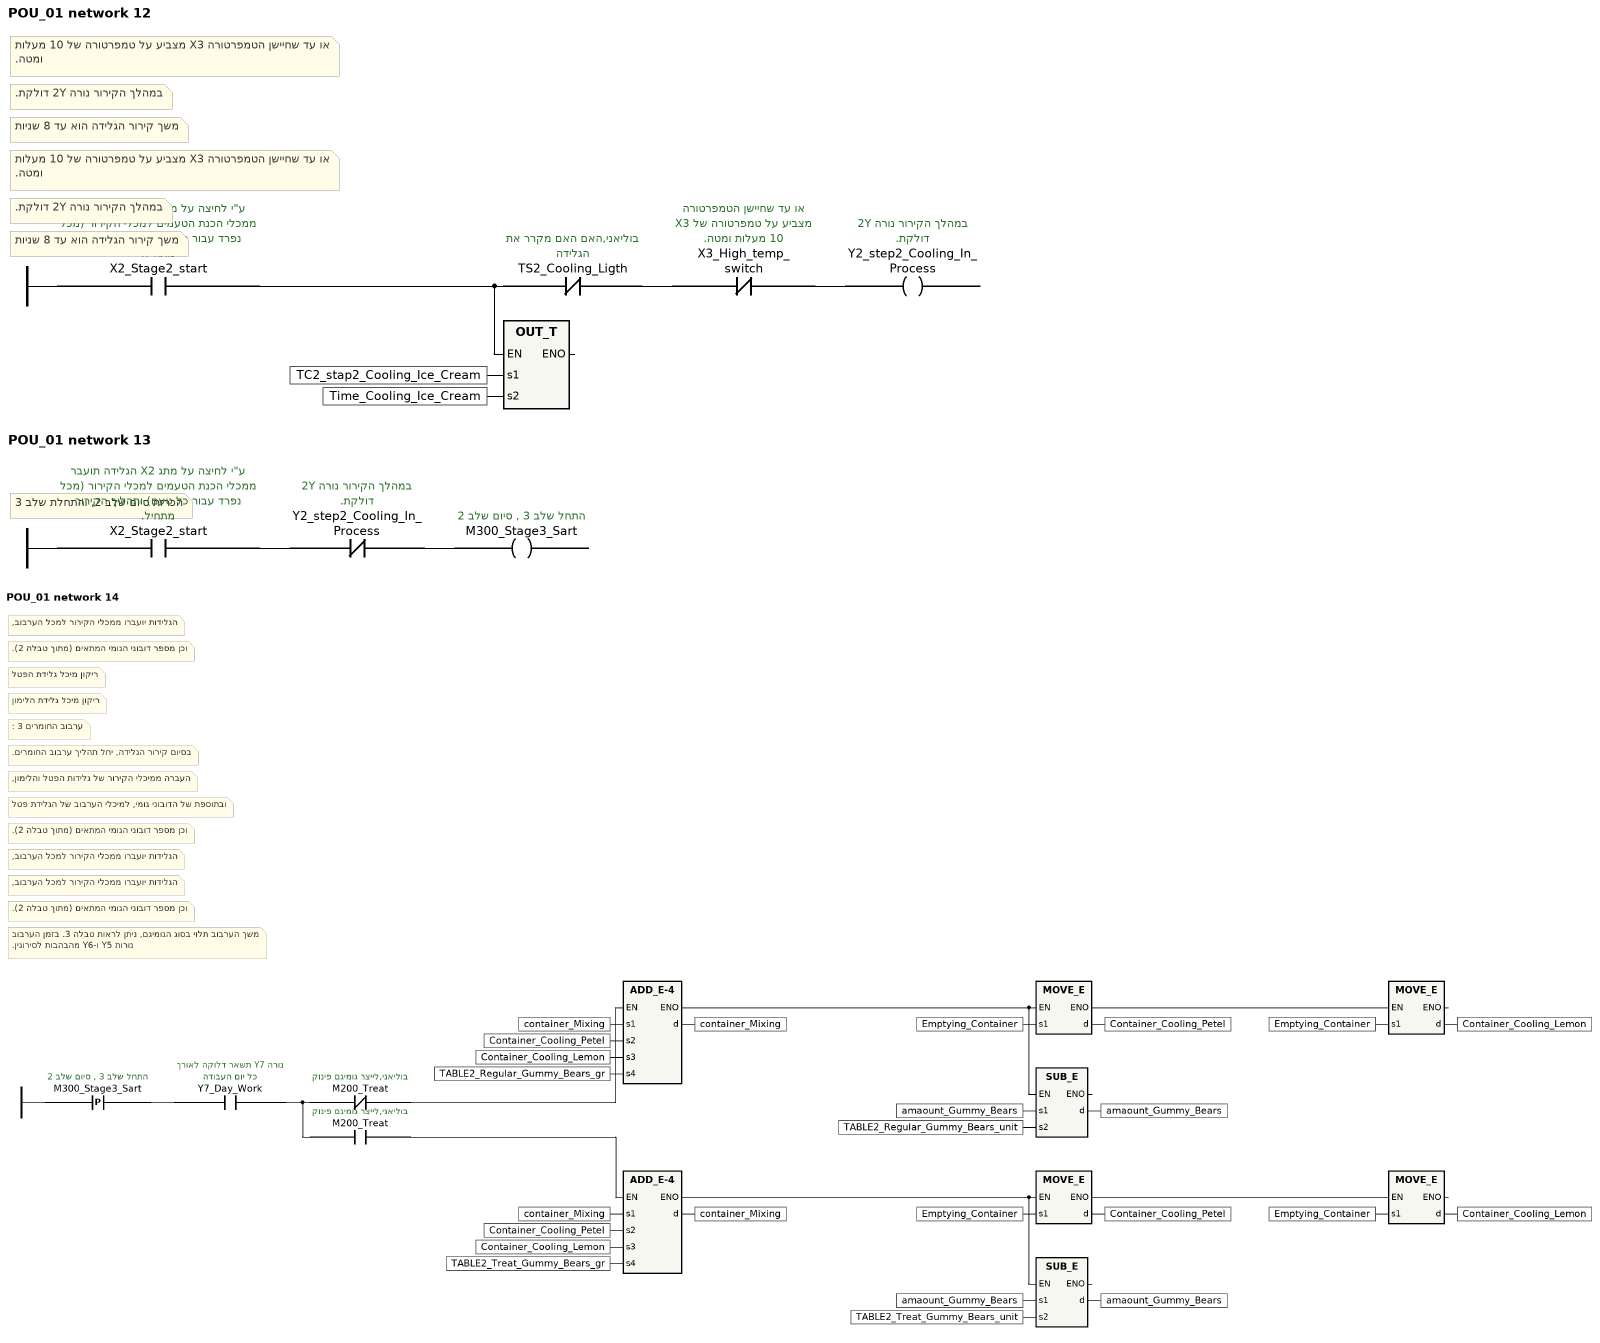
(* network 12 *)
(* או עד שחיישן הטמפרטורה X3 מצביע על טמפרטורה של 10 מעלות ומטה. *)
(* במהלך הקירור נורה 2Y דולקת. *)
(* משך קירור הגלידה הוא עד 8 שניות *)
(* או עד שחיישן הטמפרטורה X3 מצביע על טמפרטורה של 10 מעלות ומטה. *)
(* במהלך הקירור נורה 2Y דולקת. *)
(* משך קירור הגלידה הוא עד 8 שניות *)
Y2_step2_Cooling_In_Process := X2_Stage2_start AND NOT TS2_Cooling_Ligth AND NOT X3_High_temp_switch;
OUT_T(X2_Stage2_start, TC2_stap2_Cooling_Ice_Cream, Time_Cooling_Ice_Cream);
(* network 13 *)
(* הכרזת סיום שלב 2, והתחלת שלב 3 *)
M300_Stage3_Sart := X2_Stage2_start AND NOT Y2_step2_Cooling_In_Process;
(* network 14 שלב 3 *)
(* הגלידות יועברו ממכלי הקירור למכל הערבוב, *)
(* וכן מספר דובוני הגומי המתאים (מתוך טבלה 2). *)
(* ריקון מיכל גלידת הפטל *)
(* ריקון מיכל גלידת הלימון *)
(* ערבוב החומרים 3 : *)
(* בסיום קירור הגלידה, יחל תהליך ערבוב החומרים. *)
(* העברה ממיכלי הקירור של גלידות הפטל והלימון, *)
(* ובתוספת של הדובוני גומי, למיכלי הערבוב של הגלידת פטל *)
(* וכן מספר דובוני הגומי המתאים (מתוך טבלה 2). *)
(* הגלידות יועברו ממכלי הקירור למכל הערבוב, *)
(* הגלידות יועברו ממכלי הקירור למכל הערבוב, *)
(* וכן מספר דובוני הגומי המתאים (מתוך טבלה 2). *)
(* משך הערבוב תלוי בסוג הגומיגם, ניתן לראות טבלה 3. בזמן הערבוב נורות Y5 ו-Y6 מהבהבות לסירוגין. *)
_p1 := LDP(TRUE, M300_Stage3_Sart) AND Y7_Day_Work;
_e2 := ADD_E(_p1 AND NOT M200_Treat, container_Mixing, Container_Cooling_Petel, Container_Cooling_Lemon, TABLE2_Regular_Gummy_Bears_gr, container_Mixing);
_e3 := MOVE_E(_e2, Emptying_Container, Container_Cooling_Petel);
MOVE_E(_e3, Emptying_Container, Container_Cooling_Lemon);
SUB_E(_e2, amaount_Gummy_Bears, TABLE2_Regular_Gummy_Bears_unit, amaount_Gummy_Bears);
_e4 := ADD_E(_p1 AND M200_Treat, container_Mixing, Container_Cooling_Petel, Container_Cooling_Lemon, TABLE2_Treat_Gummy_Bears_gr, container_Mixing);
_e5 := MOVE_E(_e4, Emptying_Container, Container_Cooling_Petel);
MOVE_E(_e5, Emptying_Container, Container_Cooling_Lemon);
SUB_E(_e4, amaount_Gummy_Bears, TABLE2_Treat_Gummy_Bears_unit, amaount_Gummy_Bears);
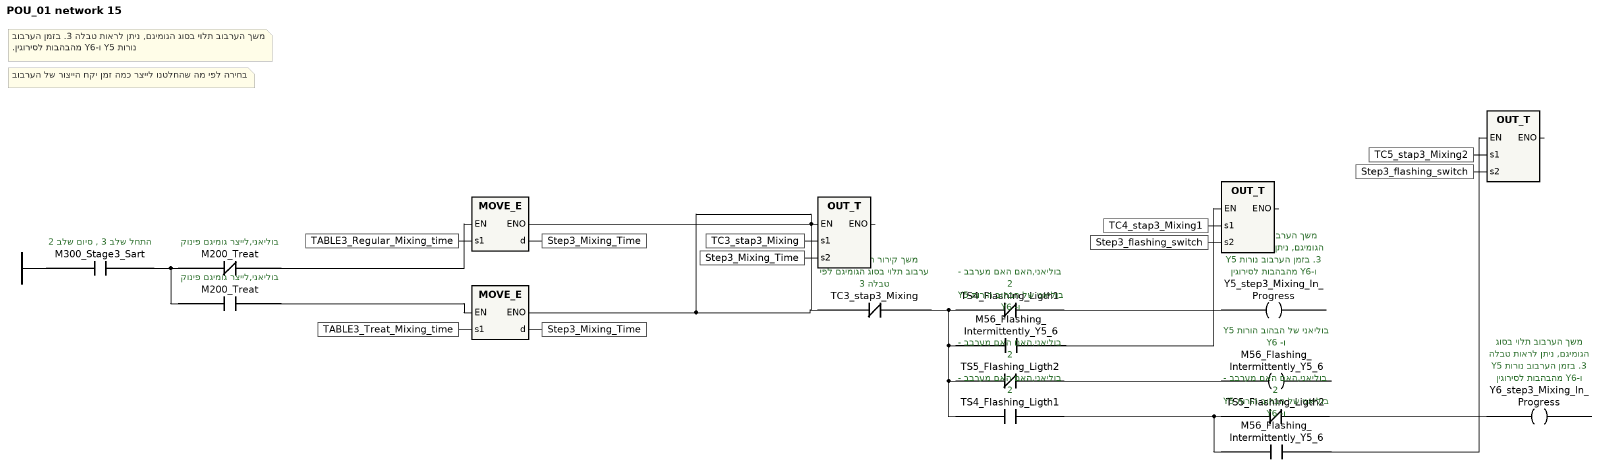
(* network 15 *)
(* משך הערבוב תלוי בסוג הגומיגם, ניתן לראות טבלה 3. בזמן הערבוב נורות Y5 ו-Y6 מהבהבות לסירוגין. *)
(* בחירה לפי מה שהחלטנו לייצר כמה זמן יקח הייצור של הערבוב *)
_e1 := MOVE_E(M300_Stage3_Sart AND NOT M200_Treat, TABLE3_Regular_Mixing_time, Step3_Mixing_Time);
_e2 := MOVE_E(M300_Stage3_Sart AND M200_Treat, TABLE3_Treat_Mixing_time, Step3_Mixing_Time);
_p3 := _e1 OR _e2;
_p4 := _p3 AND NOT TC3_stap3_Mixing;
Y5_step3_Mixing_In_Progress := _p4 AND NOT TS4_Flashing_Ligth1;
OUT_T(_p4 AND M56_Flashing_Intermittently_Y5_6, TC4_stap3_Mixing1, Step3_flashing_switch);
M56_Flashing_Intermittently_Y5_6 := _p4 AND NOT TS5_Flashing_Ligth2;
OUT_T(_p3, TC3_stap3_Mixing, Step3_Mixing_Time);
_p5 := _p4 AND TS4_Flashing_Ligth1;
Y6_step3_Mixing_In_Progress := _p5 AND NOT TS5_Flashing_Ligth2;
OUT_T(_p5 AND M56_Flashing_Intermittently_Y5_6, TC5_stap3_Mixing2, Step3_flashing_switch);
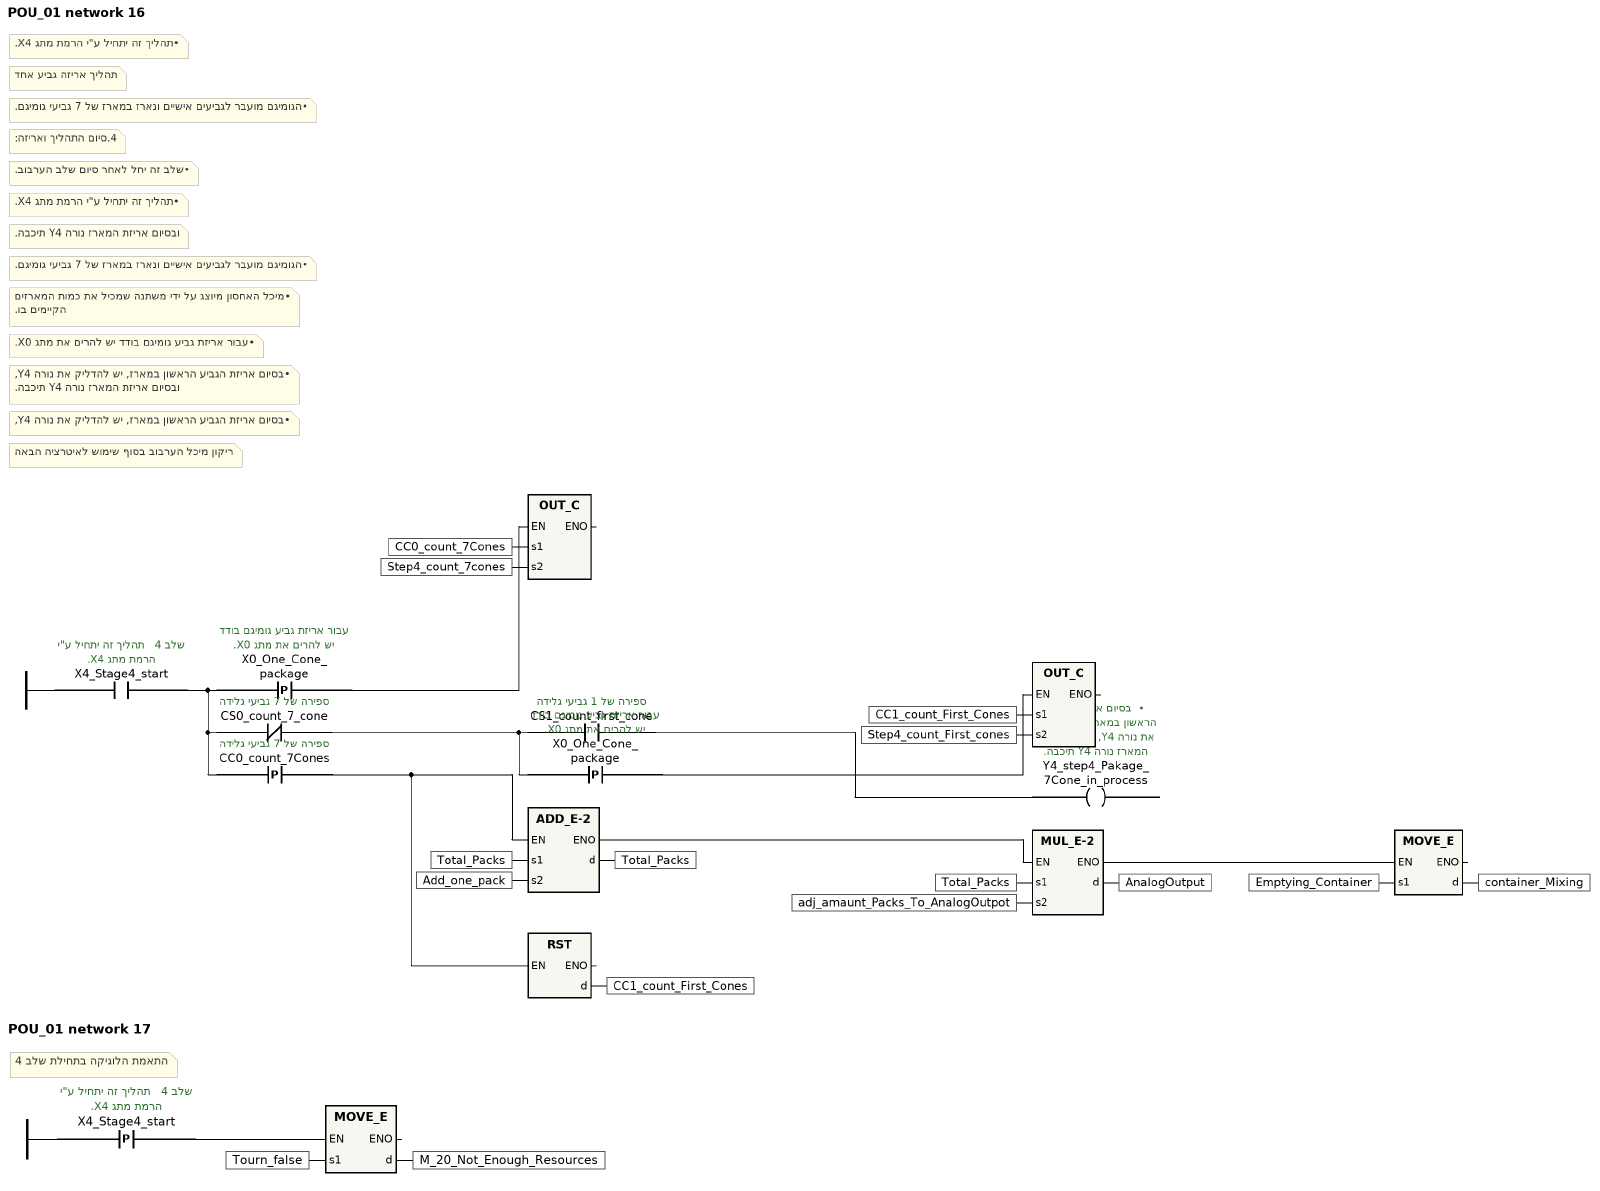
(* network 16 *)
(* •תהליך זה יתחיל ע"י הרמת מתג X4. *)
(* תהליך אריזה גביע אחד *)
(* •הגומיגם מועבר לגביעים אישיים ונארז במארז של 7 גביעי גומיגם. *)
(* 4.סיום התהליך ואריזה: *)
(* •שלב זה יחל לאחר סיום שלב הערבוב. *)
(* •תהליך זה יתחיל ע"י הרמת מתג X4. *)
(* ובסיום אריזת המארז נורה Y4 תיכבה. *)
(* •הגומיגם מועבר לגביעים אישיים ונארז במארז של 7 גביעי גומיגם. *)
(* •מיכל האחסון מיוצג על ידי משתנה שמכיל את כמות המארזים הקיימים בו. *)
(* •עבור אריזת גביע גומיגם בודד יש להרים את מתג X0. *)
(* •בסיום אריזת הגביע הראשון במארז, יש להדליק את נורה Y4, ובסיום אריזת המארז נורה Y4 תיכבה. *)
(* •בסיום אריזת הגביע הראשון במארז, יש להדליק את נורה Y4, *)
(* ריקון מיכל הערבוב בסוף שימוש לאיטרציה הבאה *)
OUT_C(X4_Stage4_start AND LDP(TRUE, X0_One_Cone_package), CC0_count_7Cones, Step4_count_7cones);
_p1 := X4_Stage4_start AND NOT CS0_count_7_cone;
Y4_step4_Pakage_7Cone_in_process := _p1 AND CS1_count_first_cone;
OUT_C(_p1 AND LDP(TRUE, X0_One_Cone_package), CC1_count_First_Cones, Step4_count_First_cones);
_p2 := X4_Stage4_start AND LDP(TRUE, CC0_count_7Cones);
RST(_p2, CC1_count_First_Cones);
_e3 := ADD_E(_p2, Total_Packs, Add_one_pack, Total_Packs);
_e4 := MUL_E(_e3, Total_Packs, adj_amaunt_Packs_To_AnalogOutpot, AnalogOutput);
MOVE_E(_e4, Emptying_Container, container_Mixing);
(* network 17 *)
(* התאמת הלוגיקה בתחילת שלב 4 *)
MOVE_E(LDP(TRUE, X4_Stage4_start), Tourn_false, M_20_Not_Enough_Resources);
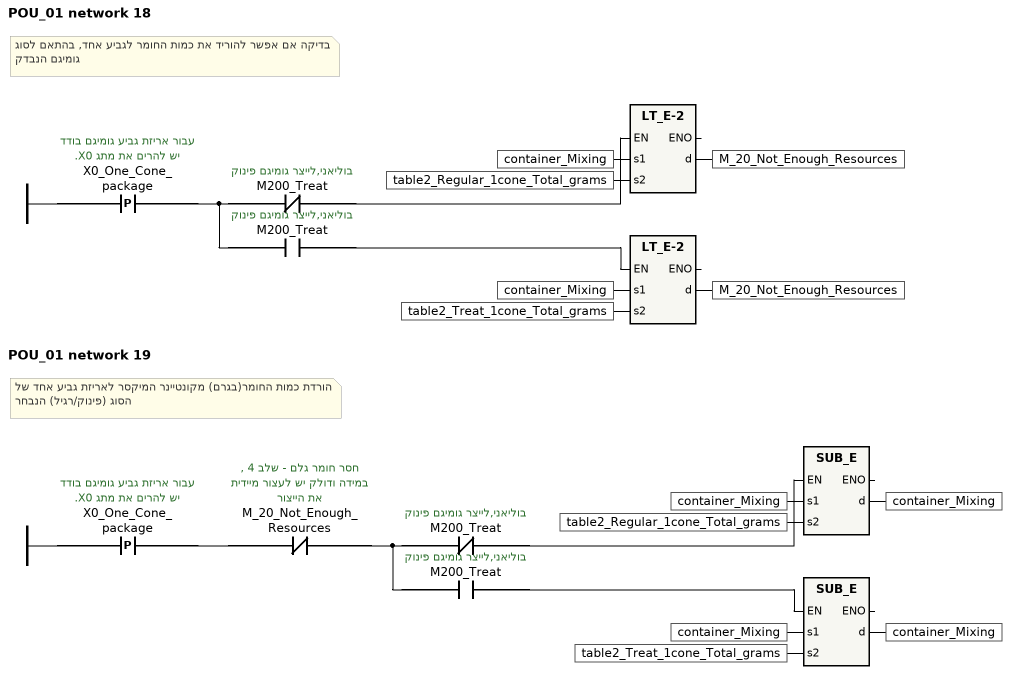
(* network 18 *)
(* בדיקה אם אפשר להוריד את כמות החומר לגביע אחד, בהתאם לסוג גומיגם הנבדק *)
_p1 := LDP(TRUE, X0_One_Cone_package);
LT_E(_p1 AND NOT M200_Treat, container_Mixing, table2_Regular_1cone_Total_grams, M_20_Not_Enough_Resources);
LT_E(_p1 AND M200_Treat, container_Mixing, table2_Treat_1cone_Total_grams, M_20_Not_Enough_Resources);
(* network 19 *)
(* הורדת כמות החומר(בגרם) מקונטיינר המיקסר לאריזת גביע אחד של הסוג (פינוק/רגיל) הנבחר *)
_p1 := LDP(TRUE, X0_One_Cone_package) AND NOT M_20_Not_Enough_Resources;
SUB_E(_p1 AND NOT M200_Treat, container_Mixing, table2_Regular_1cone_Total_grams, container_Mixing);
SUB_E(_p1 AND M200_Treat, container_Mixing, table2_Treat_1cone_Total_grams, container_Mixing);
END_PROGRAM
